FUNCTION_BLOCK conveyorHFB
  (* Standard: 61499-2 *)
  (* Version 0.1, 2017-00-12, hpea485, UOA *)
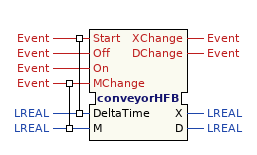
  EVENT_INPUT
    Start WITH DeltaTime;
    Off;
    On;
    MChange WITH M;
  END_EVENT
  EVENT_OUTPUT
    XChange;
    DChange;
  END_EVENT
  VAR_INPUT
    DeltaTime : LREAL;
    M : LREAL;
  END_VAR
  VAR_OUTPUT
    X : LREAL;
    D : LREAL;
  END_VAR
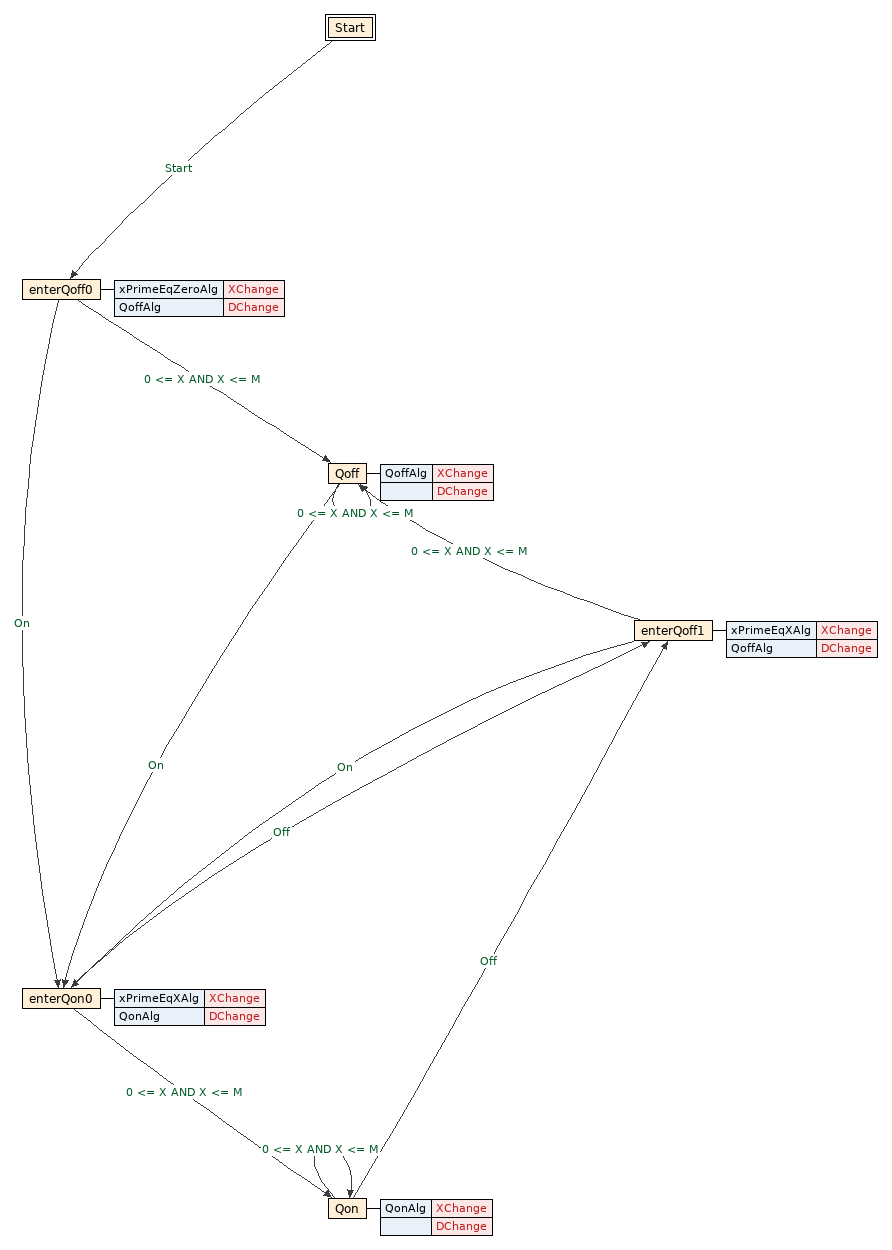
  EC_STATES
    Start;
    Qoff : QoffAlg -> XChange, -> DChange;
    Qon : QonAlg -> XChange, -> DChange;
    enterQon0 : xPrimeEqXAlg -> XChange, QonAlg -> DChange;
    enterQoff0 : xPrimeEqZeroAlg -> XChange, QoffAlg -> DChange;
    enterQoff1 : xPrimeEqXAlg -> XChange, QoffAlg -> DChange;
  END_STATES
  EC_TRANSITIONS
    Start TO enterQoff0 := Start;
    Qoff TO enterQon0 := On;
    Qoff TO Qoff := 0 <= X AND X <= M;
    Qon TO enterQoff1 := Off;
    Qon TO Qon := 0 <= X AND X <= M;
    enterQon0 TO enterQoff1 := Off;
    enterQon0 TO Qon := 0 <= X AND X <= M;
    enterQoff0 TO enterQon0 := On;
    enterQoff0 TO Qoff := 0 <= X AND X <= M;
    enterQoff1 TO enterQon0 := On;
    enterQoff1 TO Qoff := 0 <= X AND X <= M;
  END_TRANSITIONS
  ALGORITHM QoffAlg IN C: (* ODE *)
X_dot = -2 * X;
D = D + X;
  END_ALGORITHM
  ALGORITHM QonAlg IN C: (* ODE *)
X_dot = (1 - X);
D = D + X;
  END_ALGORITHM
  ALGORITHM xPrimeEqZeroAlg IN C: (* ODE_init *)
X_prime = 0;
D = 0;
  END_ALGORITHM
  ALGORITHM xPrimeEqXAlg IN C: (* ODE_init *)
X_prime = X;
D = D;
  END_ALGORITHM
END_FUNCTION_BLOCK
